{attribute 'linkalways'} 
{attribute 'no_explicit_call' := 'This FB is a CLASS and must be accessed using methods or properties'}
{attribute 'enable_dynamic_creation'}
FUNCTION_BLOCK Node_F_VN_AddToContainerElements_LREAL EXTENDS VisionNode
VAR
    fValue : _LREAL(0.0);
    ipContainer : _ITcVnContainer;
    hrPrev : _HRESULT(S_OK);
    hresult : _HRESULT(S_OK);
END_VAR

METHOD PUBLIC  Clone : I_Node
VAR
    pNode : POINTER TO Node_F_VN_AddToContainerElements_LREAL;
END_VAR
pNode := __NEW(Node_F_VN_AddToContainerElements_LREAL);
Clone := pNode^;
END_METHOD

METHOD FB_init : BOOL
VAR_INPUT
    bInitRetains : BOOL; // if TRUE, the retain variables are initialized (warm start / cold start)
    bInCopyCode : BOOL;  // if TRUE, the instance afterwards gets moved into the copy code (online change)
END_VAR
AddInput('fValue', fValue);
AddInput('ipContainer', ipContainer);
AddInput('hrPrev', hrPrev);
AddOutput('ipContainer', ipContainer);
AddOutput('hresult',hresult);
END_METHOD

METHOD PROTECTED OnExecute : HRESULT
hresult.Value := F_VN_AddToContainerElements_LREAL(
    fValue := fValue.Value,
    ipContainer := ipContainer.Value,
    hrPrev:= hrPrev.Value);
END_METHOD

METHOD PUBLIC PreExecutionCheck
VAR_INPUT
    Check : I_PreExecutionChecks;
END_VAR
Check.IsTrue(ipContainer.IsValid, 'ipContainer must be a valid container');
Check.IsTrue(ipContainer.HasType(TC_GLOBAL_CONST_LIST.ContainerType_Vector_LREAL), 'ipContainer contains incorrect type');
END_METHOD

END_FUNCTION_BLOCK

(* stored: Version 1.1.0.1, ProductVersion 3.1.4024.13
   POU Node_F_VN_AddToContainerElements_LREAL: Id {d7a8bed7-92b7-4fdd-945e-e3f544dc7d65}, SpecialFunc None
   Folder Constructor: Id {06c0ff2e-865c-41bf-b2ee-98681977027c}
   Method Clone: Id {232378fe-ee83-487e-9c9a-4566948378e5}
   Method FB_init: Id {c46f4fc3-0d0e-4cdc-8c54-539aa3903aeb}
   Method OnExecute: Id {b8af6660-c668-4742-b21b-1f4c252c4ff6}
   Method PreExecutionCheck: Id {21ad7889-5189-47e4-a355-bb89159349e6} *)
